        // -----------------------------------------------------------------
        // === STATE_HOMING (15) ===
        // -----------------------------------------------------------------
        15: // HOMING (sequential: X then Z in active homing mode 3)
            #StatusID := 2;
            // Ensure other stop/homing triggers are not interfering
            IF #homeSeqState = 1 THEN
                // Homing X
                #bHomeXExec := TRUE;
                #bHomeZExec := FALSE;
                IF #fbHomeX.Done THEN
                    #bHomeXExec := FALSE;
                    #homeSeqState := 2;    // proceed to homing Z
                    #bHomeZExec := TRUE;
                ELSIF #fbHomeX.Error THEN
                    #bHomeXExec := FALSE;
                    #bHomeZExec := FALSE;
                    #State := STATE_ERROR;
                    #newErrorFlag := TRUE;
                    #newErrorCode := 16#0003;
                    "DB_Diagnostic".HomeX_ErrorID := #fbHomeX.ErrorID;
                    "DB_Diagnostic".TO_ErrorText  := "FC_TO_ErrorText"(Code := #fbHomeX.ErrorID);
                    "DB_HMI".ErrorText      := 'Homing failed: X axis';
                    "DB_HMI".ErrorText_ES   := 'Fallo de referenciado: Eje X';
                    "DB_HMI".ErrorDetail    := CONCAT(IN1 := 'TO:', IN2 := "DB_Diagnostic".TO_ErrorText);
                    "DB_HMI".ErrorDetail_ES := CONCAT(IN1 := 'TO:', IN2 := "DB_Diagnostic".TO_ErrorText);
                END_IF;
            ELSIF #homeSeqState = 2 THEN
                // Homing Z
                #bHomeXExec := FALSE;
                #bHomeZExec := TRUE;
                IF #fbHomeZ.Done THEN
                    #bHomeZExec := FALSE;
                    IF NOT "DB_MachineConfig".Bypass_ToolAxis THEN
                        // Proceed to tool axis homing (step 3)
                        #homeSeqState := 3;
                        #bHomeToolExec := TRUE;
                    ELSE
                        // Tool axis bypassed -- go to post-homing clearance
                        #homeSeqState := 0;
                        #bHomeClrX := TRUE; #bHomeClrZ := TRUE;
                        #CurrentTool := 1;  // Tool axis homed to slot 1 position
                        #State := STATE_POST_HOME_CLR;
                    END_IF;
                ELSIF #fbHomeZ.Error THEN
                    #bHomeZExec := FALSE;
                    #State := STATE_ERROR;
                    #newErrorFlag := TRUE;
                    #newErrorCode := 16#0004;
                    "DB_Diagnostic".HomeZ_ErrorID := #fbHomeZ.ErrorID;
                    "DB_Diagnostic".TO_ErrorText  := "FC_TO_ErrorText"(Code := #fbHomeZ.ErrorID);
                    "DB_HMI".ErrorText      := 'Homing failed: Z axis';
                    "DB_HMI".ErrorText_ES   := 'Fallo de referenciado: Eje Z';
                    "DB_HMI".ErrorDetail    := CONCAT(IN1 := 'TO:', IN2 := "DB_Diagnostic".TO_ErrorText);
                    "DB_HMI".ErrorDetail_ES := CONCAT(IN1 := 'TO:', IN2 := "DB_Diagnostic".TO_ErrorText);
                END_IF;
            ELSIF #homeSeqState = 3 THEN
                // Homing Tool axis
                #bHomeToolExec := TRUE;
                IF #fbHomeTool.Done THEN
                    #bHomeToolExec := FALSE;
                    #homeSeqState := 0;
                    // Tool done -- proceed to post-homing clearance for X and Z
                    #bHomeClrX := TRUE; #bHomeClrZ := TRUE;
                    #CurrentTool := 1;  // Tool axis homed to slot 1 position
                    #State := STATE_POST_HOME_CLR;
                ELSIF #fbHomeTool.Error THEN
                    #bHomeToolExec := FALSE;
                    #State := STATE_ERROR;
                    #newErrorFlag := TRUE;
                    #newErrorCode := 16#0007;
                    "DB_Diagnostic".HomeTool_ErrorID := #fbHomeTool.ErrorID;
                    "DB_Diagnostic".TO_ErrorText     := "FC_TO_ErrorText"(Code := #fbHomeTool.ErrorID);
                    "DB_HMI".ErrorText      := 'Homing failed: Tool axis';
                    "DB_HMI".ErrorText_ES   := 'Fallo de referenciado: Eje herramienta';
                    "DB_HMI".ErrorDetail    := CONCAT(IN1 := 'TO:', IN2 := "DB_Diagnostic".TO_ErrorText);
                    "DB_HMI".ErrorDetail_ES := CONCAT(IN1 := 'TO:', IN2 := "DB_Diagnostic".TO_ErrorText);
                END_IF;
            ELSE
                // Fallback: if homeSeqState not set, go to STARTING check
                #homeSeqState := 0;
                #State := STATE_STARTING;
            END_IF;
            // Homing timeout: X+Z+Tool combined must complete within 120s
            IF #tonHomingTimeout.Q THEN
                #bHomeXExec := FALSE;
                #bHomeZExec := FALSE;
                #bHomeToolExec := FALSE;
                #homeSeqState := 0;
                #State := STATE_ERROR;
                #newErrorFlag := TRUE;
                #newErrorCode := 16#000B;
                "DB_HMI".ErrorText      := 'Homing timeout (120s)';
                "DB_HMI".ErrorText_ES   := 'Tiempo de referenciado excedido (120s)';
                "DB_HMI".ErrorDetail    := 'Homing did not complete - check reference switch/drive';
                "DB_HMI".ErrorDetail_ES := 'Referenciado no completado - revisar sensor/variador';
            END_IF;

        // -----------------------------------------------------------------
        // === STATE_PRE_HOME_CLR (13) ===
        // -----------------------------------------------------------------
        13: // PRE_HOME_CLR -- Clear PNP zone before homing
            #StatusID := 2;
            // Transition to homing as soon as clearance move finishes
            IF (NOT #bHomeClrX OR #fbMoveX_HomeClr.Done) AND (NOT #bHomeClrZ OR #fbMoveZ_HomeClr.Done) THEN
                #bHomeClrX := FALSE; #bHomeClrZ := FALSE;
                #homeSeqState := 1; #bHomeXExec := TRUE; #bHomeZExec := FALSE;
                #State := STATE_HOMING;
            ELSIF (#bHomeClrX AND #fbMoveX_HomeClr.Error) OR (#bHomeClrZ AND #fbMoveZ_HomeClr.Error) THEN
                #bHomeClrX := FALSE; #bHomeClrZ := FALSE;
                #newErrorFlag := TRUE; #newErrorCode := 16#0001;
                "DB_HMI".ErrorText      := 'Pre-home clearance move failed';
                "DB_HMI".ErrorText_ES   := 'Fallo al liberar zona PNP (pre-referencia)';
                "DB_HMI".ErrorDetail    := 'Axis could not clear PNP zone before homing - check drive';
                "DB_HMI".ErrorDetail_ES := 'Eje no pudo liberar zona PNP antes del referenciado - revisar variador';
                #State := STATE_ERROR;
            END_IF;

        // -----------------------------------------------------------------
        // === STATE_POST_HOME_CLR (16) ===
        // -----------------------------------------------------------------
        16: // POST_HOME_CLR -- Move away from PNP zone after homing
            #StatusID := 2;
            IF (NOT #bHomeClrX OR #fbMoveX_HomeClr.Done) AND (NOT #bHomeClrZ OR #fbMoveZ_HomeClr.Done) THEN
                #bHomeClrX := FALSE; #bHomeClrZ := FALSE;
                // Homing done: wait for sheet insertion before engaging ToolHeadLock
                #bSheetWaitPhase2 := FALSE;  // Always start in phase 1 (show prompt)
                #State := STATE_SHEET_WAIT;
            ELSIF (#bHomeClrX AND #fbMoveX_HomeClr.Error) OR (#bHomeClrZ AND #fbMoveZ_HomeClr.Error) THEN
                #bHomeClrX := FALSE; #bHomeClrZ := FALSE;
                #newErrorFlag := TRUE; #newErrorCode := 16#0001;
                "DB_HMI".ErrorText      := 'Post-home clearance move failed';
                "DB_HMI".ErrorText_ES   := 'Fallo al liberar zona PNP (post-referencia)';
                "DB_HMI".ErrorDetail    := 'Axis could not move from PNP zone after homing - check drive';
                "DB_HMI".ErrorDetail_ES := 'Eje no pudo salir de zona PNP despues del referenciado - revisar variador';
                #State := STATE_ERROR;
            END_IF;

        // -----------------------------------------------------------------
        // === STATE_SHEET_WAIT (14) ===
        // Phase 1: SheetHolder extends to hold the form; HMI prompt; wait operator
        //          both-button confirm (Cmd_Start rising edge).
        // Phase 2: MandrelLock extends (open-loop T#5S) to clamp the mandrel.
        // Phase 3: SheetHolder retracts (open-loop T#5S) to clear; then → LOCK_EXTEND_WAIT
        //          so ToolHeadLock engages before RUNNING.
        // -----------------------------------------------------------------
        14: // SHEET_WAIT
            #StatusID := 14;
            IF NOT #bSheetWaitPhase2 AND NOT #bSheetWaitPhase3 THEN
                // Phase 1: extend SheetHolder and prompt operator to insert the sheet
                "DB_Cylinder_SheetHolder".Cmd_Extend := TRUE;
                "DB_HMI".HasWarning     := TRUE;
                "DB_HMI".WarningText    := 'Insert sheet, then press both start buttons';
                "DB_HMI".WarningText_ES := 'Inserte la lamina y presione ambos botones de inicio';
                IF #fbInputs.Cmd_Start THEN
                    // Operator confirmed — clear prompt and begin MandrelLock extension
                    "DB_HMI".HasWarning     := FALSE;
                    "DB_HMI".WarningText    := '';
                    "DB_HMI".WarningText_ES := '';
                    "DB_Cylinder_MandrelLock".Cmd_Extend := TRUE;
                    #bSheetWaitPhase2 := TRUE;
                END_IF;
            ELSIF #bSheetWaitPhase2 THEN
                // Phase 2: open-loop wait T#5S for MandrelLock full stroke
                // tonMandrelWait is driven by the global timer section below (IN when state=14 AND phase2)
                IF #tonMandrelWait.Q THEN
                    // MandrelLock assumed clamped — retract SheetHolder
                    "DB_Cylinder_SheetHolder".Cmd_Extend := FALSE;
                    #bSheetHolderRetractPulse := TRUE;  // Force FB out of State 3 → spring retracts
                    #bSheetWaitPhase2 := FALSE;
                    #bSheetWaitPhase3 := TRUE;
                END_IF;
            ELSE
                // Phase 3: open-loop wait T#5S for SheetHolder to fully retract
                // tonSheetHolderRetract driven by global timer section below (IN when state=14 AND phase3)
                IF #tonSheetHolderRetract.Q THEN
                    #State := STATE_LOCK_EXTEND_WAIT;  // ToolHeadLock engages, then → RUNNING
                END_IF;
            END_IF;

        // -----------------------------------------------------------------
        // === STATE_RUNNING (20) ===
        // -----------------------------------------------------------------
        20: // RUNNING
            #StatusID := 3; #bStartSeq := TRUE;
            #timerRunning := TRUE;  // Start cycle timer

            // Update HMI
            "DB_HMI".CurrentLine := #fbRecipeHandler.CurrentLine;
            "DB_HMI".ProgressPercent := #fbRecipeHandler.Progress;
            "DB_HMI".FeedrateActive := #fbRecipeHandler.ActiveFeedrate;

            IF #bPauseActive THEN #State := STATE_PAUSED; END_IF;

            // Tool change request (bypass if no tool axis)
            IF #fbRecipeHandler.ToolChangeReq THEN
                IF "DB_MachineConfig".Bypass_ToolAxis THEN
                    // Skip tool change - clear request and continue
                    #fbRecipeHandler.ToolChangeReq := FALSE;
                ELSIF #fbRecipeHandler.ToolReqNumber = #CurrentTool THEN
                    // Requested tool already in position (e.g. home = slot 1) - skip retract/rotate/extend
                    #fbRecipeHandler.ToolChangeReq := FALSE;
                ELSE
                    #activeToolReq    := #fbRecipeHandler.ToolReqNumber;
                    #bStartSeq        := FALSE;
                    // Release lock before rotating turret: wait T#2S in LOCK_RETRACT_WAIT,
                    // then proceed to STATE_TOOL_CHANGE.
                    #bLockAfterHoming := FALSE;  // LOCK_RETRACT_WAIT exits to STATE_TOOL_CHANGE
                    #State            := STATE_LOCK_RETRACT_WAIT;
                END_IF;
            END_IF;

            // Spindle control from recipe
            IF #fbRecipeHandler.SpindleReqStart THEN
                IF #bSpindleDecelWait THEN
                    // Decel timer still running — capture for deferred apply
                    #bSpindlePendingStart := TRUE;
                    #pendingSpindleSpeed  := #fbRecipeHandler.SpindleReqSpeed;
                ELSE
                    #bSpindleStart := TRUE;
                    "DB_Spindle".Cmd_SetSpeed := #fbRecipeHandler.SpindleReqSpeed;
                END_IF;
            END_IF;
            IF #fbRecipeHandler.SpindleReqStop THEN
                #bSpindleStart       := FALSE;  // Drop RunCmd level
                #bSpindleDecelWait   := TRUE;   // Start decel wait
                #bSpindlePendingStart := FALSE; // Cancel any previous pending start
            END_IF;

            // Complete
            IF #fbRecipeHandler.Done THEN
                #State := 100;  // Go to COMPLETE state, not IDLE
                "DB_HMI".ProgressPercent := 100.0;
                #bSpindleStart := FALSE;  // Drop RunCmd level on completion
                #timerRunning := FALSE; // Stop cycle timer
                #savedLineIndex := -1;  // Clear saved position
                #savedProgram := -1;
            END_IF;

            // Error
            IF #fbRecipeHandler.Error THEN
                #State := STATE_ERROR;
                #newErrorFlag := TRUE;
                #newErrorCode := #fbRecipeHandler.ErrorID;
            END_IF;

        // -----------------------------------------------------------------
        // === STATE_LOCK_EXTEND_WAIT (17) ===
        // -----------------------------------------------------------------
        17: // LOCK_EXTEND_WAIT -- commanding ToolHeadLock to extend; sensor must confirm before RUNNING
            // Cmd_Extend=TRUE is driven outside the CASE (see ToolHeadLock section below).
            // No timer fallback -- lock MUST be confirmed by sensor before machining starts.

 	     #StatusID := 17;
	      IF "DB_Cylinder_ToolHeadLock".AtSetpoint THEN
 	         #State := STATE_RUNNING;
 	     ELSIF "DB_Cylinder_ToolHeadLock".Error THEN
  	        // Sensor did not confirm within Timeout_Extend (T#3S) — abort
  	        #newErrorFlag := TRUE;
  	        #newErrorCode := 16#0012;
  	        "DB_HMI".ErrorText      := 'ToolHeadLock: extend timeout';
  	        "DB_HMI".ErrorText_ES   := 'Bloqueo cabezal: tiempo de extension excedido';
   	       "DB_HMI".ErrorDetail    := 'Lock sensor (AtSetpoint) not confirmed - check cylinder/sensor';
   	       "DB_HMI".ErrorDetail_ES := 'Sensor de bloqueo (AtSetpoint) no confirmado - revisar cilindro/sensor';
   	       #State := STATE_ERROR;
   	   END_IF;

        // -----------------------------------------------------------------
        // === STATE_LOCK_RETRACT_WAIT (29) ===
        // -----------------------------------------------------------------
        29: // LOCK_RETRACT_WAIT -- ToolHeadLock releasing (spring return); wait T#2S before proceeding
            // Cmd_Extend=FALSE here (state not RUNNING/PAUSED/LOCK_EXTEND_WAIT); spring retracts.
            // No sensor yet: proceed after timeout regardless.
            // bLockAfterHoming selects exit:
            //   TRUE  = coming from STOPPING → go to STATE_STOP_GOHOME (homing after stop)
            //   FALSE = coming from RUNNING (tool change) → go to STATE_TOOL_CHANGE
            #StatusID := 29;
            IF #tonLockWait.Q THEN
                IF #bLockAfterHoming THEN
                    #homeSeqState := 1;
                    #bHomeXExec   := TRUE;
                    #State        := STATE_STOP_GOHOME;
                ELSE
                    #State := STATE_TOOL_CHANGE;
                END_IF;
            END_IF;

        // -----------------------------------------------------------------
        // === STATE_STOPPING (18) ===
        // -----------------------------------------------------------------
        18: // STOPPING - Stop program without generating an error; then home all axes.
            // After recipe executor finishes, spindle is stopped and all axes are homed
            // (X → Z → Tool, same sequence as STATE_HOMING) so the machine is at a known
            // reference position ready for the next run or manual mode.
            #StatusID := 18;
            #Running := FALSE;
            #timerRunning := FALSE;
            // Phase 1: wait for recipe executor to finish, then command spindle stop and
            // begin waiting for the spindle to reach zero speed before releasing MandrelLock.
            // MandrelLock stays extended (sheet clamped) while the spindle decelerates --
            // retracting while spinning could throw the sheet at the operator.
            IF NOT #fbRecipeHandler.Busy AND NOT #bWaitingSpindleStop THEN
                #bSpindleStop             := TRUE;
                #bSheetHolderRetractPulse := TRUE;  // One-shot: release sheet holder (may be extended if stopped during SHEET_WAIT Ph1/2)
                #bSheetWaitPhase2         := FALSE;
                #bSheetWaitPhase3         := FALSE;
                #bWaitingSpindleStop      := TRUE;  // Enable phase 2 (spindle zero-speed check)
            END_IF;
            // Phase 2: release MandrelLock once spindle decel timer has elapsed.
            // No physical encoder on spindle axis -- ActualSpeed is a TO estimate only.
            // Timer (tonSpindleStopWait T#10S) is the sole release condition.
            IF #bWaitingSpindleStop AND #tonSpindleStopWait.Q THEN
                "DB_Cylinder_MandrelLock".Cmd_Extend := FALSE;
                #bMandrelRetractPulse  := TRUE;  // One-shot: release mandrel lock
                #bWaitingSpindleStop   := FALSE;
                #bLockAfterHoming      := TRUE;  // LOCK_RETRACT_WAIT exits to STATE_STOP_GOHOME
                #State                 := STATE_LOCK_RETRACT_WAIT;
            END_IF;

        // -----------------------------------------------------------------
        // === STATE_STOP_GOHOME (19) ===
        // -----------------------------------------------------------------
        19: // STOP_GOHOME - Active homing after stop (X then Z, sequential)
            // BUG FIX: Previous implementation homed X and Z simultaneously.
            // Using the same sequential pattern as STATE_HOMING: X first, then Z.
            #StatusID := 19;
            #Running := FALSE;
            IF #homeSeqState = 1 THEN
                // X homing
                #bHomeXExec := TRUE;
                #bHomeZExec := FALSE;
                IF #fbHomeX.Done THEN
                    #bHomeXExec := FALSE;
                    #homeSeqState := 2;
                    #bHomeZExec := TRUE;
                ELSIF #fbHomeX.Error THEN
                    #bHomeXExec := FALSE;
                    #homeSeqState := 0;
                    #State := STATE_ERROR;
                    #newErrorFlag := TRUE;
                    #newErrorCode := 16#0003;
                    "DB_Diagnostic".HomeX_ErrorID := #fbHomeX.ErrorID;
                    "DB_Diagnostic".TO_ErrorText  := "FC_TO_ErrorText"(Code := #fbHomeX.ErrorID);
                    "DB_HMI".ErrorText      := 'Post-stop homing failed: X';
                    "DB_HMI".ErrorText_ES   := 'Fallo de referenciado post-paro: X';
                    "DB_HMI".ErrorDetail    := CONCAT(IN1 := 'TO:', IN2 := "DB_Diagnostic".TO_ErrorText);
                    "DB_HMI".ErrorDetail_ES := CONCAT(IN1 := 'TO:', IN2 := "DB_Diagnostic".TO_ErrorText);
                END_IF;
            ELSIF #homeSeqState = 2 THEN
                // Z homing
                #bHomeXExec := FALSE;
                #bHomeZExec := TRUE;
                IF #fbHomeZ.Done THEN
                    #bHomeZExec := FALSE;
                    IF NOT "DB_MachineConfig".Bypass_ToolAxis THEN
                        // Proceed to tool axis homing (step 3)
                        #homeSeqState := 3;
                        #bHomeToolExec := TRUE;
                    ELSE
                        // Tool axis bypassed -- homing complete
                        #homeSeqState := 0;
                        #State := STATE_STOPPED;
                    END_IF;
                ELSIF #fbHomeZ.Error THEN
                    #bHomeZExec := FALSE;
                    #homeSeqState := 0;
                    #State := STATE_ERROR;
                    #newErrorFlag := TRUE;
                    #newErrorCode := 16#0004;
                    "DB_Diagnostic".HomeZ_ErrorID := #fbHomeZ.ErrorID;
                    "DB_Diagnostic".TO_ErrorText  := "FC_TO_ErrorText"(Code := #fbHomeZ.ErrorID);
                    "DB_HMI".ErrorText      := 'Post-stop homing failed: Z';
                    "DB_HMI".ErrorText_ES   := 'Fallo de referenciado post-paro: Z';
                    "DB_HMI".ErrorDetail    := CONCAT(IN1 := 'TO:', IN2 := "DB_Diagnostic".TO_ErrorText);
                    "DB_HMI".ErrorDetail_ES := CONCAT(IN1 := 'TO:', IN2 := "DB_Diagnostic".TO_ErrorText);
                END_IF;
            ELSIF #homeSeqState = 3 THEN
                // Homing Tool axis
                #bHomeToolExec := TRUE;
                IF #fbHomeTool.Done THEN
                    #bHomeToolExec := FALSE;
                    #homeSeqState := 0;
                    #State := STATE_STOPPED;
                ELSIF #fbHomeTool.Error THEN
                    #bHomeToolExec := FALSE;
                    #homeSeqState := 0;
                    #State := STATE_ERROR;
                    #newErrorFlag := TRUE;
                    #newErrorCode := 16#0007;
                    "DB_Diagnostic".HomeTool_ErrorID := #fbHomeTool.ErrorID;
                    "DB_Diagnostic".TO_ErrorText     := "FC_TO_ErrorText"(Code := #fbHomeTool.ErrorID);
                    "DB_HMI".ErrorText      := 'Post-stop homing failed: Tool';
                    "DB_HMI".ErrorText_ES   := 'Fallo de referenciado post-paro: Herramienta';
                    "DB_HMI".ErrorDetail    := CONCAT(IN1 := 'TO:', IN2 := "DB_Diagnostic".TO_ErrorText);
                    "DB_HMI".ErrorDetail_ES := CONCAT(IN1 := 'TO:', IN2 := "DB_Diagnostic".TO_ErrorText);
                END_IF;
            ELSE
                // homeSeqState invalid -- safe fallback
                #homeSeqState := 0;
                #bHomeXExec := FALSE;
                #bHomeZExec := FALSE;
                #bHomeToolExec := FALSE;
                #State := STATE_STOPPED;
            END_IF;
            // Homing timeout: X+Z+Tool combined must complete within 120s
            IF #tonHomingTimeout.Q THEN
                #bHomeXExec := FALSE;
                #bHomeZExec := FALSE;
                #bHomeToolExec := FALSE;
                #homeSeqState := 0;
                #State := STATE_ERROR;
                #newErrorFlag := TRUE;
                #newErrorCode := 16#000B;
                "DB_HMI".ErrorText      := 'Homing timeout (120s)';
                "DB_HMI".ErrorText_ES   := 'Tiempo de referenciado excedido (120s)';
                "DB_HMI".ErrorDetail    := 'Post-stop homing did not complete - check reference switch/drive';
                "DB_HMI".ErrorDetail_ES := 'Referenciado post-paro no completado - revisar sensor/variador';
            END_IF;

        // -----------------------------------------------------------------
        // === STATE_STOP_GOTOZERO (21) ===
        // -----------------------------------------------------------------
        21: // STOP_GOTOZERO - Go to position 0 after stop
            #StatusID := 21;
            #Running := FALSE;
            // Has X axis motion completed?
            IF #bStopMoveX AND #fbMoveX_Stop.Done THEN
                #bStopMoveX := FALSE;
            ELSIF #bStopMoveX AND #fbMoveX_Stop.Error THEN
                #bStopMoveX := FALSE;
                #State := STATE_ERROR;
                #newErrorFlag := TRUE;
                #newErrorCode := 16#0001; // X move failed
                "DB_HMI".ErrorText      := 'Post-stop X move failed';
                "DB_HMI".ErrorText_ES   := 'Fallo de movimiento post-paro: X';
                "DB_HMI".ErrorDetail    := 'X axis could not return to zero after stop';
                "DB_HMI".ErrorDetail_ES := 'Eje X no pudo retornar a cero despues del paro';
            END_IF;
            // Has Z axis motion completed?
            IF #bStopMoveZ AND #fbMoveZ_Stop.Done THEN
                #bStopMoveZ := FALSE;
            ELSIF #bStopMoveZ AND #fbMoveZ_Stop.Error THEN
                #bStopMoveZ := FALSE;
                #State := STATE_ERROR;
                #newErrorFlag := TRUE;
                #newErrorCode := 16#0002; // Z move failed
                "DB_HMI".ErrorText      := 'Post-stop Z move failed';
                "DB_HMI".ErrorText_ES   := 'Fallo de movimiento post-paro: Z';
                "DB_HMI".ErrorDetail    := 'Z axis could not return to zero after stop';
                "DB_HMI".ErrorDetail_ES := 'Eje Z no pudo retornar a cero despues del paro';
            END_IF;
            // When both axes are done, return to STOPPED
            IF NOT #bStopMoveX AND NOT #bStopMoveZ AND (#State = STATE_STOP_GOTOZERO) THEN
                #State := STATE_STOPPED;
            END_IF;

        // -----------------------------------------------------------------
        // === STATE_PNP_HALT (22) ===
        // -----------------------------------------------------------------
        22: // PNP_HALT -- axis halted at proximity zone; drives ON, reverse jog allowed to escape
            #StatusID := 22;
            #Running := FALSE;
            // Auto-exit: PNP zone cleared (axis has moved away) -- return to STOPPED
            IF NOT #HW_PNP_X_Min AND NOT #HW_PNP_X_Max THEN #bHaltX_PNP := FALSE; END_IF;
            IF NOT #HW_PNP_Z_Min AND NOT #HW_PNP_Z_Max THEN #bHaltZ_PNP := FALSE; END_IF;
            IF NOT #bHaltX_PNP AND NOT #bHaltZ_PNP THEN
                #State := STATE_STOPPED;
            END_IF;
            // Manual exit: operator presses AckError or Reset
            IF (#ackEdge OR #fbInputs.Cmd_Reset) AND (#EStop_OK OR "DB_HMI".Bypass_EStop) THEN
                #bHaltX_PNP := FALSE;
                #bHaltZ_PNP := FALSE;
                #Error := FALSE;
                #prevSafetyError := FALSE;
                #fbAlarmManager(NewError := FALSE, NewErrorCode := 0, AcknowledgeError := TRUE);
                #State := STATE_STOPPED;
            END_IF;
            // Forward spindle commands from recipe handler.
            // When PNP fires during STATE_RUNNING, the RUNNING(20) case is skipped, so
            // bSpindleStart is never updated from fbRecipeHandler signals. Mirror them here.
            // Note: fbRecipeHandler runs AFTER this CASE, so values here are from previous scan.
            IF #fbRecipeHandler.SpindleReqStop THEN
                #bSpindleStart := FALSE;  // Drop RunCmd level
            END_IF;
            IF #fbRecipeHandler.SpindleReqStart THEN
                #bSpindleStart := TRUE;
                "DB_Spindle".Cmd_SetSpeed := #fbRecipeHandler.SpindleReqSpeed;
            END_IF;

        // -----------------------------------------------------------------
        // === STATE_PAUSED (25) ===
        // -----------------------------------------------------------------
        25: // PAUSED
            #StatusID := 88;
            // Stop elapsed time counting while paused
            #timerRunning := FALSE;
            // Only Btn_Continue resumes (Pause button does NOT toggle)
            IF #continueEdge THEN
                #bPauseActive := FALSE;
                #State := STATE_RUNNING;
            END_IF;

        // -----------------------------------------------------------------
        // === STATE_TOOL_CHANGE (30) ===
        // -----------------------------------------------------------------
        30: // TOOL_CHANGE
            #StatusID := 4; #bToolExecute := TRUE; #State := STATE_TOOL_WAIT;

        // -----------------------------------------------------------------
        // === STATE_TOOL_WAIT (35) ===
        // -----------------------------------------------------------------
        35: // TOOL_WAIT
            IF #fbToolChanger.Done THEN
                #bToolExecute := FALSE;
                #CurrentTool := #fbToolChanger.CurrentTool;
                #fbRecipeHandler.ToolChangeReq := FALSE;  // Signal RecipeHandler to continue
                // Tool change done: re-engage lock before resuming machining
                #State := STATE_LOCK_EXTEND_WAIT;
            ELSIF #fbToolChanger.Error THEN
                #bToolExecute := FALSE;
                #State := STATE_ERROR;
                #newErrorFlag := TRUE;
                #newErrorCode := #fbToolChanger.ErrorID;
                "DB_HMI".ErrorText      := 'Tool changer failed';
                "DB_HMI".ErrorText_ES   := 'Fallo en cambiador de herramienta';
                "DB_HMI".ErrorDetail    := CONCAT(IN1 := 'Tool ', IN2 := INT_TO_STRING(#activeToolReq));
                "DB_HMI".ErrorDetail_ES := CONCAT(IN1 := 'Herramienta ', IN2 := INT_TO_STRING(#activeToolReq));
            END_IF;

        // -----------------------------------------------------------------
        // === STATE_ERROR (999) ===
        // -----------------------------------------------------------------
        999: // ERROR
            #StatusID := 99; #bStartSeq := FALSE; #Error := TRUE;
            #timerRunning := FALSE;  // Stop cycle timer
            // Clear CMD=41 BackSupport overrides — valves de-energise on error
            "DB_Cylinder_BackSupport".SolB_Cmd41  := FALSE;
            "DB_Cylinder_BackSupport".SolAtmo_Cmd := FALSE;
            // SheetHolder: clear extend command while in error so it does not hold on reset
            "DB_Cylinder_SheetHolder".Cmd_Extend  := FALSE;

            // Save current position for warm restart
            IF #savedLineIndex < 0 THEN
                #savedLineIndex := #fbRecipeHandler.CurrentLine;
                #savedProgram := #activeProgram;
            END_IF;
            "DB_HMI".ResumeLine := #savedLineIndex;   // HMI shows which line will be resumed on next Start

            // Debug: populate DB_Diagnostic with error context for easier troubleshooting
            "DB_Diagnostic".Error_ProcessState := #State;
            "DB_Diagnostic".Error_Code := #fbAlarmManager.ActiveErrorCode; // primary error source
            // If recipe handler provided an error line, prefer that
            IF "DB_Diagnostic".Recipe_CurrentLine >= 0 THEN
                "DB_Diagnostic".Error_Line := "DB_Diagnostic".Recipe_CurrentLine;
            END_IF;

            // BUG FIX: Previous implementation transitioned ackEdge → STATE_PAUSED,
            // but the recipe handler remained in its internal STATE_ERROR (999).
            // In PAUSED → Continue → STATE_RUNNING the recipe handler was not running (error state).
            // Fix: All recovery paths go to STATE_STOPPED + recipe handler is reset.
            // When operator presses Start, PRE_SCAN → STARTING → RUNNING flow starts clean.
            // ACK, Continue and Restart are blocked while E-Stop is active.
            // E-Stop must be physically released before any error acknowledgement is accepted.
            IF #ackEdge AND (#EStop_OK OR "DB_HMI".Bypass_EStop) THEN
                // Acknowledge: clear error → STOPPED. savedLineIndex kept for warm restart on next Start.
                #Error := FALSE;
                #bPauseActive := FALSE;
                #bResetRecipe := TRUE;   // Reset recipe handler to IDLE (cannot continue from state 999)
                #prevSafetyError := FALSE;   // Clear safety latch -- fresh evaluation on restart
                #bSheetWaitPhase2         := FALSE;
                #bSheetWaitPhase3         := FALSE;
                #bMandrelRetractPulse     := TRUE;  // Release mandrel lock (may be extended from last run)
                #bSheetHolderRetractPulse := TRUE;  // Release sheet holder (may be extended from last run)
                #fbAlarmManager(NewError := FALSE, NewErrorCode := 0,
                                AcknowledgeError := TRUE);
                #State := STATE_STOPPED;
            ELSIF #continueEdge AND (#EStop_OK OR "DB_HMI".Bypass_EStop) THEN
                // Continue: resume from savedLineIndex on next Start (warm restart)
                #Error := FALSE;
                #bPauseActive := FALSE;
                #bResetRecipe := TRUE;
                #bSheetWaitPhase2         := FALSE;
                #bSheetWaitPhase3         := FALSE;
                #bMandrelRetractPulse     := TRUE;  // Release mandrel lock
                #bSheetHolderRetractPulse := TRUE;  // Release sheet holder
                #fbAlarmManager(NewError := FALSE, NewErrorCode := 0,
                                AcknowledgeError := TRUE);
                #State := STATE_STOPPED;
            ELSIF #restartEdge AND (#EStop_OK OR "DB_HMI".Bypass_EStop) THEN
                // Restart: explicit restart from line 0 -- clear saved position
                #Error := FALSE;
                #bPauseActive := FALSE;
                #bResetRecipe := TRUE;
                #savedLineIndex := -1;
                #savedProgram := -1;
                "DB_HMI".ResumeLine := -1;
                #bSheetWaitPhase2         := FALSE;
                #bSheetWaitPhase3         := FALSE;
                #bMandrelRetractPulse     := TRUE;  // Release mandrel lock
                #bSheetHolderRetractPulse := TRUE;  // Release sheet holder
                #fbAlarmManager(NewError := FALSE, NewErrorCode := 0,
                                AcknowledgeError := TRUE);
                #State := STATE_STOPPED;
            END_IF;
    END_CASE;

    // -----------------------------------------------------------------
    // === STATE_COMPLETE (100) ===
    // (handled as IF block outside CASE -- no new constant needed)
    // -----------------------------------------------------------------
    IF #State = 100 THEN
        #StatusID := 100; #bStartSeq := FALSE;
        #Running := FALSE;
        // Clear bSpindleStart: RUNNING no longer runs to clear it, so SpindleReqStart=TRUE
        // from the last CMD_SPINDLE_ON would keep Start=TRUE through PRE_SCAN and STARTING.
        // prevStart is reset inside FB_SpindleControl on halt Done, so the next CMD_SPINDLE_ON
        // in the new recipe generates a clean startEdge.
        // bSpindleStop is intentionally NOT cleared here: line 1567 sets it TRUE on Done to
        // stop the spindle, and clearing it in the same scan (IF State=100 runs same scan as
        // the Done handler in CASE 20) would cancel the stop command before it is consumed.
        #bSpindleStart := FALSE;
        "DB_Cylinder_MandrelLock".Cmd_Extend := FALSE;
        #bMandrelRetractPulse := TRUE;          // One-shot: force mandrel lock FB out of State 3 → spring retracts
        "DB_Cylinder_BackSupport".SolB_Cmd41  := FALSE;  // De-energise CMD=41 Sol_B override
        "DB_Cylinder_BackSupport".SolAtmo_Cmd := FALSE;  // De-energise atmosphere valve
        "DB_HMI".StatusMsg    := 'Program Complete';
        "DB_HMI".StatusMsg_ES := 'Programa Completado';
        "DB_HMI".ErrorText    := 'Done!';
        "DB_HMI".ErrorText_ES := '¡Completado!';
        IF #fbInputs.Cmd_Start OR #restartEdge THEN
            "DB_HMI".CycleCount := "DB_HMI".CycleCount + 1;
            #bResetRecipe := TRUE;      // Reset FB_RecipeHandler (state 99→0) before re-run
            #State := STATE_PRE_SCAN;   // Restart/Start = immediate re-run, keeps drives on
        ELSIF #fbInputs.Cmd_Reset THEN
            "DB_HMI".CycleCount := "DB_HMI".CycleCount + 1;
            #bResetRecipe := TRUE;      // Also reset recipe handler on manual reset
            #State := STATE_PRE_SCAN;    // Reset from COMPLETE goes to PRE_SCAN (drives stay on)
        END_IF;
    END_IF;

    // =========================================================================
    // CYCLE TIMER - runs during RUNNING and PAUSED
    // =========================================================================
    #tonElapsed(IN := #timerRunning, PT := T#24h);
    // Homing timeout: counts only while in a homing state; auto-resets when state exits
    #tonHomingTimeout(IN := (#State = STATE_HOMING OR #State = STATE_STOP_GOHOME), PT := T#120S);
    // ToolHeadLock wait: counts in both lock wait states; auto-resets on exit
    // tonLockWait: 5s total (1s pre-delay + up to 4s for cylinder stroke). AtSetpoint exits early.
    #tonLockWait(IN := (#State = STATE_LOCK_RETRACT_WAIT),
                 PT := T#5S);  // Retract wait only -- no fallback for extend (sensor required)
    #tonLockPreDelay(IN := (#State = STATE_LOCK_EXTEND_WAIT), PT := T#1S);
    // Spindle-stop wait: safety fallback for MandrelLock retract in STATE_STOPPING.
    // Starts when phase 2 begins (bWaitingSpindleStop); fires after 5s if ActualSpeed never drops.
    #tonSpindleStopWait(IN := (#State = STATE_STOPPING AND #bWaitingSpindleStop), PT := T#10S);
    // MandrelLock stroke wait: open-loop T#5S during STATE_SHEET_WAIT phase 2
    #tonMandrelWait(IN := (#State = STATE_SHEET_WAIT AND #bSheetWaitPhase2), PT := T#5S);
    // SheetHolder retract wait: open-loop T#5S during STATE_SHEET_WAIT phase 3
    #tonSheetHolderRetract(IN := (#State = STATE_SHEET_WAIT AND #bSheetWaitPhase3), PT := T#5S);
    // One-shot retract pulses:
    // ValveType=1 + Mode=0 keeps Sol_A=TRUE in State 3 even after Cmd_Extend=FALSE.
    // A one-scan Cmd_Retract=TRUE pulse forces the FB to State 2 (Sol_A=FALSE) → spring retracts.
    "DB_Cylinder_MandrelLock".Cmd_Retract  := #bMandrelRetractPulse;
    #bMandrelRetractPulse := FALSE;  // Self-clearing: active for exactly one scan
    "DB_Cylinder_SheetHolder".Cmd_Retract  := #bSheetHolderRetractPulse;
    #bSheetHolderRetractPulse := FALSE;  // Self-clearing: active for exactly one scan
    // Drive ready timeout: counts while in STARTING and drives not yet ready; auto-resets on exit
    #tonDriveReady(IN := (#State = STATE_STARTING) AND NOT (#fbPowerX.Status AND #fbPowerZ.Status), PT := T#3S);
    // Spindle decel wait: blocks RunCmd from going TRUE until VFD ramp-down completes
    #tonSpindleDecel(IN := #bSpindleDecelWait, PT := "DB_MachineConfig".SpindleDecelTime);
    IF #tonSpindleDecel.Q THEN
        #bSpindleDecelWait := FALSE;
        IF #bSpindlePendingStart THEN
            "DB_Spindle".Cmd_SetSpeed := #pendingSpindleSpeed;
            #bSpindleStart        := TRUE;
            #bSpindlePendingStart := FALSE;
        END_IF;
    END_IF;
    IF #timerRunning THEN
        "DB_HMI".ElapsedTime := #tonElapsed.ET;
        "DB_HMI".ElapsedSeconds := TIME_TO_DINT(#tonElapsed.ET / 1000);
    END_IF;
    // Reset timer on new program start
    IF #State = STATE_STARTING THEN
        #tonElapsed(IN := FALSE, PT := T#24h);  // Reset
        "DB_HMI".ElapsedTime := T#0s;
        "DB_HMI".ElapsedSeconds := 0;
    END_IF;

    // =========================================================================
    // PRODUCTION LOGGING - DB_Production
    // =========================================================================
    // Edge: cycle start (enter PRE_SCAN)
    IF (#State = STATE_PRE_SCAN) AND (#prevState <> STATE_PRE_SCAN) THEN
        "DB_Production".CurrentActive := TRUE;
        "DB_Production".CurrentProgram := #activeProgram;
        "DB_Production".TotalStarted := "DB_Production".TotalStarted + 1;
        #prodTimeStatus := RD_SYS_T(OUT => #prodTimeNow);
        "DB_Production".CurrentStartTime := #prodTimeNow;
    END_IF;

    // Edge: OK complete (enter state 100)
    IF (#State = 100) AND (#prevState <> 100) THEN
        "DB_Production".LastResult := 1;  // OK
        "DB_Production".LastProgram := #activeProgram;
        "DB_Production".LastDuration_s := "DB_HMI".ElapsedSeconds;
        "DB_Production".LastErrorCode := 0;
        "DB_Production".LastErrorLine := -1;
        "DB_Production".TotalOK := "DB_Production".TotalOK + 1;
        #prodTimeStatus := RD_SYS_T(OUT => #prodTimeNow);
        "DB_Production".LastEndTime := #prodTimeNow;
        "DB_Production".CurrentActive := FALSE;

        // History ring buffer update
        "DB_Production".Hist_Index := "DB_Production".Hist_Index + 1;
        IF "DB_Production".Hist_Index > 100 THEN
            "DB_Production".Hist_Index := 1;
        END_IF;
        IF "DB_Production".Hist_Count < 100 THEN
            "DB_Production".Hist_Count := "DB_Production".Hist_Count + 1;
        END_IF;
        "DB_Production".Hist_Result["DB_Production".Hist_Index] := "DB_Production".LastResult;
        "DB_Production".Hist_Program["DB_Production".Hist_Index] := "DB_Production".LastProgram;
        "DB_Production".Hist_Duration_s["DB_Production".Hist_Index] := "DB_Production".LastDuration_s;
        "DB_Production".Hist_ErrorCode["DB_Production".Hist_Index] := "DB_Production".LastErrorCode;
        "DB_Production".Hist_ErrorLine["DB_Production".Hist_Index] := "DB_Production".LastErrorLine;
        "DB_Production".Hist_Time["DB_Production".Hist_Index] := #prodTimeNow;
    END_IF;

    // Edge: NOK (enter STATE_ERROR with active cycle)
    IF (#State = STATE_ERROR) AND (#prevState <> STATE_ERROR) AND "DB_Production".CurrentActive THEN
        "DB_Production".LastResult := 2;  // NOK
        "DB_Production".LastProgram := #activeProgram;
        "DB_Production".LastDuration_s := "DB_HMI".ElapsedSeconds;
        "DB_Production".LastErrorCode := #fbAlarmManager.ActiveErrorCode;
        "DB_Production".LastErrorLine := "DB_Diagnostic".Error_Line;
        "DB_Production".TotalNOK := "DB_Production".TotalNOK + 1;
        #prodTimeStatus := RD_SYS_T(OUT => #prodTimeNow);
        "DB_Production".LastEndTime := #prodTimeNow;
        "DB_Production".CurrentActive := FALSE;

        // History ring buffer update
        "DB_Production".Hist_Index := "DB_Production".Hist_Index + 1;
        IF "DB_Production".Hist_Index > 100 THEN
            "DB_Production".Hist_Index := 1;
        END_IF;
        IF "DB_Production".Hist_Count < 100 THEN
            "DB_Production".Hist_Count := "DB_Production".Hist_Count + 1;
        END_IF;
        "DB_Production".Hist_Result["DB_Production".Hist_Index] := "DB_Production".LastResult;
        "DB_Production".Hist_Program["DB_Production".Hist_Index] := "DB_Production".LastProgram;
        "DB_Production".Hist_Duration_s["DB_Production".Hist_Index] := "DB_Production".LastDuration_s;
        "DB_Production".Hist_ErrorCode["DB_Production".Hist_Index] := "DB_Production".LastErrorCode;
        "DB_Production".Hist_ErrorLine["DB_Production".Hist_Index] := "DB_Production".LastErrorLine;
        "DB_Production".Hist_Time["DB_Production".Hist_Index] := #prodTimeNow;
    END_IF;

    // Edge: STOPPED via STOP sequence (STOPPING / STOP_GOHOME / STOP_GOTOZERO → STOPPED)
    IF (#State = STATE_STOPPED) AND
       ((#prevState = STATE_STOPPING) OR (#prevState = STATE_STOP_GOHOME) OR (#prevState = STATE_STOP_GOTOZERO)) AND
       "DB_Production".CurrentActive THEN
        "DB_Production".LastResult := 3;  // STOP
        "DB_Production".LastProgram := #activeProgram;
        "DB_Production".LastDuration_s := "DB_HMI".ElapsedSeconds;
        "DB_Production".LastErrorCode := 0;
        "DB_Production".LastErrorLine := -1;
        "DB_Production".TotalStopped := "DB_Production".TotalStopped + 1;
        #prodTimeStatus := RD_SYS_T(OUT => #prodTimeNow);
        "DB_Production".LastEndTime := #prodTimeNow;
        "DB_Production".CurrentActive := FALSE;

        // History ring buffer update
        "DB_Production".Hist_Index := "DB_Production".Hist_Index + 1;
        IF "DB_Production".Hist_Index > 100 THEN
            "DB_Production".Hist_Index := 1;
        END_IF;
        IF "DB_Production".Hist_Count < 100 THEN
            "DB_Production".Hist_Count := "DB_Production".Hist_Count + 1;
        END_IF;
        "DB_Production".Hist_Result["DB_Production".Hist_Index] := "DB_Production".LastResult;
        "DB_Production".Hist_Program["DB_Production".Hist_Index] := "DB_Production".LastProgram;
        "DB_Production".Hist_Duration_s["DB_Production".Hist_Index] := "DB_Production".LastDuration_s;
        "DB_Production".Hist_ErrorCode["DB_Production".Hist_Index] := "DB_Production".LastErrorCode;
        "DB_Production".Hist_ErrorLine["DB_Production".Hist_Index] := "DB_Production".LastErrorLine;
        "DB_Production".Hist_Time["DB_Production".Hist_Index] := #prodTimeNow;
    END_IF;

    // Production RESET: clear counters + history
    IF #prodResetEdge THEN
        "DB_Production".TotalStarted := 0;
        "DB_Production".TotalOK := 0;
        "DB_Production".TotalNOK := 0;
        "DB_Production".TotalStopped := 0;
        "DB_Production".Hist_Index := 0;
        "DB_Production".Hist_Count := 0;
        // Optionally also clear last cycle summary
        "DB_Production".LastResult := 0;
        "DB_Production".LastProgram := 0;
        "DB_Production".LastDuration_s := 0;
        "DB_Production".LastErrorCode := 0;
        "DB_Production".LastErrorLine := -1;
        "DB_Production".CurrentActive := FALSE;
    END_IF;

    // Last-cycle RESET: only clear last cycle summary (counters and history are preserved)
    IF #lastCycleResetEdge THEN
        "DB_Production".LastResult := 0;
        "DB_Production".LastProgram := 0;
        "DB_Production".LastDuration_s := 0;
        "DB_Production".LastErrorCode := 0;
        "DB_Production".LastErrorLine := -1;
    END_IF;

    // Update prevState for next cycle
    #prevState := #State;

    // =========================================================================
    // RECIPE HANDLER - Execute based on active program
    // =========================================================================
    CASE #activeProgram OF
        1: #fbRecipeHandler(Start := #bStartSeq, Stop := #fbInputs.Cmd_Stop,
                            Pause := #bPauseActive, Reset := #fbInputs.Cmd_Reset OR #bResetRecipe,
                            bStartEdge := #fbInputs.Cmd_Start,
                            StartLine := MAX(IN1:= INT#0, IN2:= #savedLineIndex),
                            LineCount := #activeLineCount,
                            Lines := "DB_RecipeProgram1".Lines,
                            Axis_X := #Axis_X, Axis_Z := #Axis_Z);
        2: #fbRecipeHandler(Start := #bStartSeq, Stop := #fbInputs.Cmd_Stop,
                            Pause := #bPauseActive, Reset := #fbInputs.Cmd_Reset OR #bResetRecipe,
                            bStartEdge := #fbInputs.Cmd_Start,
                            StartLine := MAX(IN1:= INT#0,IN2:= #savedLineIndex),
                            LineCount := #activeLineCount,
                            Lines := "DB_RecipeProgram2".Lines,
                            Axis_X := #Axis_X, Axis_Z := #Axis_Z);
        3: #fbRecipeHandler(Start := #bStartSeq, Stop := #fbInputs.Cmd_Stop,
                            Pause := #bPauseActive, Reset := #fbInputs.Cmd_Reset OR #bResetRecipe,
                            bStartEdge := #fbInputs.Cmd_Start,
                            StartLine := MAX(IN1:= INT#0,IN2:= #savedLineIndex),
                            LineCount := #activeLineCount,
                            Lines := "DB_RecipeProgram3".Lines,
                            Axis_X := #Axis_X, Axis_Z := #Axis_Z);
        4: #fbRecipeHandler(Start := #bStartSeq, Stop := #fbInputs.Cmd_Stop,
                            Pause := #bPauseActive, Reset := #fbInputs.Cmd_Reset OR #bResetRecipe,
                            bStartEdge := #fbInputs.Cmd_Start,
                            StartLine := MAX(IN1:= INT#0,IN2:= #savedLineIndex),
                            LineCount := #activeLineCount,
                            Lines := "DB_RecipeProgram4".Lines,
                            Axis_X := #Axis_X, Axis_Z := #Axis_Z);
        5: #fbRecipeHandler(Start := #bStartSeq, Stop := #fbInputs.Cmd_Stop,
                            Pause := #bPauseActive, Reset := #fbInputs.Cmd_Reset OR #bResetRecipe,
                            bStartEdge := #fbInputs.Cmd_Start,
                            StartLine := MAX(IN1:= INT#0,IN2:= #savedLineIndex),
                            LineCount := #activeLineCount,
                            Lines := "DB_RecipeProgram5".Lines,
                            Axis_X := #Axis_X, Axis_Z := #Axis_Z);
    END_CASE;

    // Homing -- sequential pattern: STATE_HOMING (startup) and STATE_STOP_GOHOME (post-stop)
    // both use homeSeqState + bHomeXExec/bHomeZExec.
    // Mode SEL: mode 3 (active+zero) is forced in STATE_HOMING; other states use DB_Manual.HomingMode.
    #fbHomeX(
        Execute := #bHomeXExec,
        Mode := SEL(G := (#State = STATE_HOMING AND #bHomeXExec), IN0 := 3, IN1 := "DB_Manual".HomingMode),
        Position := "DB_MachineConfig".HomeOffset_X,
        Axis := #Axis_X
    );
    #fbHomeZ(
        Execute := #bHomeZExec,
        Mode := SEL(G := (#State = STATE_HOMING AND #bHomeZExec), IN0 := 3, IN1 := "DB_Manual".HomingMode),
        Position := "DB_MachineConfig".HomeOffset_Z,
        Axis := #Axis_Z
    );
    #fbHomeTool(
        Execute  := #bHomeToolExec,
        Mode     := SEL(G := (#State = STATE_HOMING AND #bHomeToolExec), IN0 := 3, IN1 := "DB_Manual".HomingMode),
        Position := 0.0,
        Axis     := #Axis_Tool
    );
    // PNP halt FBs: Execute stays TRUE until bHaltX/Z_PNP is cleared (on return to STATE_STOPPED)
    #fbHaltX_PNP(Execute := #bHaltX_PNP, Axis := #Axis_X);
    #fbHaltZ_PNP(Execute := #bHaltZ_PNP, Axis := #Axis_Z);

    // Tool changer -- only rotates the turret; axis positioning done by G-code
    #fbToolChanger(Execute := #bToolExecute, ToolNumber := #activeToolReq,
                   Axis_Tool := #Axis_Tool);

    // Motion FBs for moving to position 0 after stop
    #fbMoveX_Stop(Execute := #bStopMoveX, Position := 0.0, Velocity := "DB_MachineConfig".RapidVelocity, Axis := #Axis_X);
    #fbMoveZ_Stop(Execute := #bStopMoveZ, Position := 0.0, Velocity := "DB_MachineConfig".RapidVelocity, Axis := #Axis_Z);
    // Homing clearance moves -- pre (clear PNP zone) and post (move away after homing)
    // Target: HomeOffset + PostHome_Clearance (outside PNP sensor range)
    #fbMoveX_HomeClr(Execute  := #bHomeClrX,
                     Position := "DB_MachineConfig".HomeOffset_X + "DB_MachineConfig".PostHome_Clearance,
                     Velocity := "DB_MachineConfig".HomeVelocity,
                     Axis     := #Axis_X);
    #fbMoveZ_HomeClr(Execute  := #bHomeClrZ,
                     Position := "DB_MachineConfig".HomeOffset_Z + "DB_MachineConfig".PostHome_Clearance,
                     Velocity := "DB_MachineConfig".HomeVelocity,
                     Axis     := #Axis_Z);

    // Manual mode - sync aliases first
    // In STATE_PNP_HALT: block jog direction that would drive the axis deeper into the PNP zone.
    // Jog toward the active PNP zone is blocked; jog away (escape direction) is passed through.
    IF #State = STATE_PNP_HALT THEN
        "DB_Manual".Jog_Plus  := "DB_Manual".Btn_JogPlus AND NOT (
            ("DB_Manual".SelectedAxis = 0 AND #HW_PNP_X_Max) OR
            ("DB_Manual".SelectedAxis = 1 AND #HW_PNP_Z_Max));
        "DB_Manual".Jog_Minus := "DB_Manual".Btn_JogMinus AND NOT (
            ("DB_Manual".SelectedAxis = 0 AND #HW_PNP_X_Min) OR
            ("DB_Manual".SelectedAxis = 1 AND #HW_PNP_Z_Min));
    ELSE
        "DB_Manual".Jog_Plus  := "DB_Manual".Btn_JogPlus;
        "DB_Manual".Jog_Minus := "DB_Manual".Btn_JogMinus;
    END_IF;
    "DB_Manual".Btn_HomeAxis := "DB_Manual".Btn_Home;

    #fbManualMode(Enable := (#State = STATE_MANUAL OR #State = STATE_PNP_HALT),
                  SelectedAxis := "DB_Manual".SelectedAxis,
                  Jog_Plus := "DB_Manual".Jog_Plus, Jog_Minus := "DB_Manual".Jog_Minus,
                  JogSpeed := "DB_Manual".JogSpeed,
                  MoveAbsolute := "DB_Manual".Btn_MoveAbsolute, TargetPosition := "DB_Manual".MoveToPosition,
                  HomeAxis := "DB_Manual".Btn_HomeAxis, HomeAll := "DB_Manual".Btn_HomeAll,
                  HomingMode := "DB_Manual".HomingMode, HomePosition := 0.0,
                  GoSafe := "DB_Manual".Btn_GoSafe, GoZero := "DB_Manual".Btn_GoZero,
                  SafeToJog := #fbSafetyMonitor.SafeToJog, Reset := #fbInputs.Cmd_Reset,
                  PNP_X_Min := #HW_PNP_X_Min, PNP_Z_Min := #HW_PNP_Z_Min,
                  ToolStepCW := "DB_Manual".Btn_ToolStepCW, ToolStepCCW := "DB_Manual".Btn_ToolStepCCW,
                  ToolStepAngle := "DB_Manual".ToolStepAngle, ToolStepSpeed := "DB_Manual".ToolStepSpeed,
                  Axis_X := #Axis_X, Axis_Z := #Axis_Z, Axis_Tool := #Axis_Tool, Axis_Spindle := #Axis_Spindle);

    // Update manual mode status
    "DB_Manual".JogBusy := #fbManualMode.Busy;
    "DB_Manual".ManualBusy := #fbManualMode.Busy;       // Alias
    "DB_Manual".JogError := #fbManualMode.Error;
    "DB_Manual".ManualError := #fbManualMode.Error;     // Alias
    "DB_Manual".JogErrorID := #fbManualMode.ErrorID;
    "DB_Manual".ManualErrorID := #fbManualMode.ErrorID; // Alias
    "DB_Manual".SelectedAxisPos := SEL(G := "DB_Manual".SelectedAxis = 0,
                                        IN0 := #Axis_Z.ActualPosition, IN1 := #Axis_X.ActualPosition);
    "DB_Manual".SelectedAxisName := SEL(G := "DB_Manual".SelectedAxis = 0, IN0 := 'Z', IN1 := 'X');
    "DB_Manual".ToolPosition := #Axis_Tool.ActualPosition;
    "DB_Manual".ActiveAxis := #fbManualMode.ActiveAxis;

    // Forward manual mode errors to alarm manager (once, on rising edge)
    IF #fbManualMode.Error AND NOT #prevManualError THEN
        #newErrorFlag := TRUE;
        #newErrorCode := #fbManualMode.ErrorID;
        // DB_HMI.ErrorDetail is written directly inside FB_ManualMode at each error point.
        // Write ErrorText here as a fallback for any code not yet handled with direct detail.
        "DB_HMI".ErrorText    := 'Manual mode error - check ErrorDetail and ErrorID';
        "DB_HMI".ErrorText_ES := 'Error modo manual - revisar ErrorDetail y ErrorID';
    END_IF;
    #prevManualError := #fbManualMode.Error;

    // =========================================================================
    // SPINDLE CONTROL
    // Manual mode spindle control via DB_Manual buttons
    // Recipe handler spindle control via bSpindleStart/bSpindleStop flags
    // =========================================================================
    // Capture inputs BEFORE calling the FB so Diag_* reflects this scan's values.
    "DB_Spindle".Diag_bSpindleStart := #bSpindleStart;
    "DB_Spindle".Diag_bSpindleStop  := #bSpindleStop;
    "DB_Spindle".Diag_EnableInput   := #bDrivesEnable;
    "DB_Spindle".Diag_StartInput    := "DB_Manual".Btn_SpindleStart OR #bSpindleStart;
    "DB_Spindle".Diag_StopInput     := "DB_Manual".Btn_SpindleStop OR #bSpindleStop OR #fbInputs.Cmd_Stop;
    "DB_Spindle".Diag_ReqStart      := #fbRecipeHandler.SpindleReqStart;
    "DB_Spindle".Diag_ReqStop       := #fbRecipeHandler.SpindleReqStop;
    // -------------------------------------------------------------------------
    // Spindle history ring buffer: push snapshot on any meaningful change.
    // Trigger fields: SpindleState, PrevStart, ReqStart, StartEdge.
    // Reading tip: sort Hist_Log[0..19] by .Seq to get chronological order.
    // -------------------------------------------------------------------------
    IF "DB_Spindle".Hist_Clear THEN
        "DB_Spindle".Hist_Head   := 0;
        "DB_Spindle".Hist_Count  := 0;
        "DB_Spindle".Hist_SeqNum := 0;
        "DB_Spindle".Hist_Clear  := FALSE;
    ELSIF ("DB_Spindle".Diag_SpindleState <> #prevSnap_State)
       OR ("DB_Spindle".Diag_PrevStart    <> #prevSnap_PrevStart)
       OR ("DB_Spindle".Diag_ReqStart     <> #prevSnap_ReqStart)
       OR ("DB_Spindle".Diag_StartEdge    <> #prevSnap_StartEdge)
       OR ("DB_Spindle".Diag_MoveVelBusy  <> #prevSnap_MoveVelBusy) THEN
        // Push new entry at Hist_Head
        "DB_Spindle".Hist_Log["DB_Spindle".Hist_Head].Seq          := "DB_Spindle".Hist_SeqNum;
        "DB_Spindle".Hist_Log["DB_Spindle".Hist_Head].MachineState := #State;
        "DB_Spindle".Hist_Log["DB_Spindle".Hist_Head].State        := "DB_Spindle".Diag_SpindleState;
        "DB_Spindle".Hist_Log["DB_Spindle".Hist_Head].ReqStart     := "DB_Spindle".Diag_ReqStart;
        "DB_Spindle".Hist_Log["DB_Spindle".Hist_Head].ReqStop      := "DB_Spindle".Diag_ReqStop;
        "DB_Spindle".Hist_Log["DB_Spindle".Hist_Head].bStart       := "DB_Spindle".Diag_bSpindleStart;
        "DB_Spindle".Hist_Log["DB_Spindle".Hist_Head].bStop        := "DB_Spindle".Diag_bSpindleStop;
        "DB_Spindle".Hist_Log["DB_Spindle".Hist_Head].StartInput   := "DB_Spindle".Diag_StartInput;
        "DB_Spindle".Hist_Log["DB_Spindle".Hist_Head].StopInput    := "DB_Spindle".Diag_StopInput;
        "DB_Spindle".Hist_Log["DB_Spindle".Hist_Head].EnableIn     := "DB_Spindle".Diag_EnableInput;
        "DB_Spindle".Hist_Log["DB_Spindle".Hist_Head].PrevStart    := "DB_Spindle".Diag_PrevStart;
        "DB_Spindle".Hist_Log["DB_Spindle".Hist_Head].StartEdge    := "DB_Spindle".Diag_StartEdge;
        "DB_Spindle".Hist_Log["DB_Spindle".Hist_Head].MoveVelBusy  := "DB_Spindle".Diag_MoveVelBusy;
        "DB_Spindle".Hist_Log["DB_Spindle".Hist_Head].MoveVelInVel := "DB_Spindle".Diag_MoveVelInVel;
        // Advance ring buffer pointer
        "DB_Spindle".Hist_SeqNum := "DB_Spindle".Hist_SeqNum + 1;
        "DB_Spindle".Hist_Head   := ("DB_Spindle".Hist_Head + 1) MOD 20;
        IF "DB_Spindle".Hist_Count < 20 THEN
            "DB_Spindle".Hist_Count := "DB_Spindle".Hist_Count + 1;
        END_IF;
        // Latch current values for next-scan comparison
        #prevSnap_State       := "DB_Spindle".Diag_SpindleState;
        #prevSnap_PrevStart   := "DB_Spindle".Diag_PrevStart;
        #prevSnap_ReqStart    := "DB_Spindle".Diag_ReqStart;
        #prevSnap_StartEdge   := "DB_Spindle".Diag_StartEdge;
        #prevSnap_MoveVelBusy := "DB_Spindle".Diag_MoveVelBusy;
    END_IF;
    // RunCmd is a level signal (TRUE = run).
    // The CALLER must:
    //   • Set SetSpeed before raising RunCmd
    //   • Lower RunCmd to stop (do not change SetSpeed while RunCmd is TRUE)
    //   • For a speed change: lower RunCmd → update SetSpeed → raise RunCmd again
    #fbSpindleControl(
        Enable   := #bDrivesEnable,
        RunCmd   := ("DB_Manual".Btn_SpindleStart OR #bSpindleStart)
                    AND NOT ("DB_Manual".Btn_SpindleStop OR #bSpindleStop OR #fbInputs.Cmd_Stop),
        SetSpeed := SEL(G := (#State = STATE_MANUAL),
                        IN0 := "DB_Spindle".Cmd_SetSpeed,
                        IN1 := "DB_Manual".Manual_SpindleSpeed),
        SpeedOverride := "DB_Spindle".SpeedOverride,
        Reset    := #fbInputs.Cmd_Reset,
        AckError := #ackEdge OR "DB_Manual".Btn_SpindleAckError,
	RunForward := "PTO_RunForward_AxisS",
        Axis_Spindle := #Axis_Spindle
    );
    // Write FB outputs back to DB_Spindle so HMI tags reflect actual state
    "DB_Spindle".IsRunning    := #fbSpindleControl.Running;
    "DB_Spindle".AtSpeed      := #fbSpindleControl.AtSpeed;
    "DB_Spindle".ActualSpeed  := #fbSpindleControl.ActualSpeed;

    // =========================================================================
    // TOOLHEADLOCK CONTROL
    // Written every scan so FB_CylinderControl (called from OB1) sees the
    // correct command on the next scan.
    //
    // EXTEND (Sol_A ON):  STATE_RUNNING (20), STATE_PAUSED (25), STATE_LOCK_EXTEND_WAIT (17)
    // RETRACT (spring):   all other states -- cylinder retracts automatically via spring return.
    //
    // Safety: spring-return valve retracts on power loss without any PLC action.
    // State 17 checks AtSetpoint for extend confirmation only -- no fallback timer in FB_Process.
    // CylFB Timeout_Extend (T#6S in DB_Cylinder_ToolHeadLock) is the sole timer; on timeout
    // CylFB sets Error=TRUE, state 17 catches it and goes to STATE_ERROR (16#0012).
    // State 29 uses tonLockWait only (spring retract; no retract sensor).
    // =========================================================================
    "DB_Cylinder_ToolHeadLock".Cmd_Extend :=
        (#State = STATE_RUNNING) OR
        (#State = STATE_PAUSED) OR
        (#State = STATE_LOCK_EXTEND_WAIT AND #tonLockPreDelay.Q);

    // Diagnostic output
    "DB_Diagnostic".Process_State        := #State;
    "DB_Diagnostic".Process_SafeToRun    := #SafeToRun;
    "DB_Diagnostic".Process_DrivesEnable := #bDrivesEnable;
    "DB_Diagnostic".Recipe_CurrentProgram := #activeProgram;
    "DB_Diagnostic".Recipe_TotalLines    := #activeLineCount;
    "DB_Diagnostic".Axis_X_Pos           := #Axis_X.ActualPosition;
    "DB_Diagnostic".Axis_Z_Pos           := #Axis_Z.ActualPosition;
    "DB_Diagnostic".Axis_X_Enabled       := #fbPowerX.Status;
    "DB_Diagnostic".Axis_Z_Enabled       := #fbPowerZ.Status;
    "DB_Diagnostic".Axis_X_Homed         := #Axis_X.StatusBits.HomingDone;
    "DB_Diagnostic".Axis_Z_Homed         := #Axis_Z.StatusBits.HomingDone;

    // =========================================================================
    // CONTACTOR CONTROL -- called as the last step of FB_Process.
    // FC_ContactorControl reads DB_HMI.Btn_Contactor_* and Bypass_EStop/HasError.
    // In auto mode STATE_STARTING already sets these flags TRUE; they are reflected to I/O here.
    // Called here rather than from OB1 to ensure contactor logic runs in sync with the process.
    // =========================================================================
    "FC_ContactorControl"();
END_FUNCTION_BLOCK
